TYPE IPC_Standard:
STRUCT
	MesData	: IPC;  (* (NA) Object	*)
END_STRUCT
END_TYPE

(* stored: Version 1.1.0.1, ProductVersion 3.1.4024.11
   DUT IPC_Standard: Id {b665ce76-6dcf-4a31-809b-590683547280} *)
